{attribute addProperty BoxType "EL6224-0000-0021"}
{attribute addProperty Id "Device_DiagAT %I*BOOL1Device_StateAT %I*BOOL1"}
{attribute addProperty CRC "2703295896"}
{attribute addProperty SizeInBites "16"}
{attribute addProperty SizeInBytes "2"}
TYPE DeviceState_Inputs_Device_A1210598 :
STRUCT
	{attribute addProperty Name "Device_Diag"}
	Device_Diag AT %I* : BOOL;
	{attribute addProperty Name "Device_State"}
	Device_State AT %I* : BOOL;
END_STRUCT
END_TYPE

(* stored: Version 1.2.0.0, ProductVersion 3.1.4024.9
   DUT DeviceState_Inputs_Device_A1210598: Id {1bd5a2ff-5163-4ca6-9263-8f51b7c9d508} *)
